{attribute 'qualified_only'}
VAR_GLOBAL
	(*IO*)
	stTest04_DigitalInput:stHMI_DigitalInput;
	stTest05_DigitalInput:stHMI_DigitalInput;
	
	(*SYSTEM*)
	stTest01_Intlk:stHMI_Interlock;
	stTest02_Perm:stHMI_Permissive;
	stTest03_RunCtrl:stHMI_SystemRunControl;
END_VAR

(* stored: Version 1.1.0.1, ProductVersion 3.1.4024.11
   GVL GVL_HMI: Id {9df10dcc-a297-45fd-afd9-0c7547cf2255} *)
